(* CODESYS project para_retain.20190301.5.project

Project tree, tasks and I/O mapping:
  MIC7001 : Changsha Xiangji-ARM Cortex A9(xilinx zynq7000)-linux, Changsha Xiangji Hiden Technology Co.Ltd, version 3.5.10.40
    application Application
      libraries: CAA Types Extern, 3.5.10.0 (CAA Technical Workgroup); VisuDialogs, * (System); CAA Real Time Clock Extern, 3.5.10.0 (CAA Technical Workgroup); CAA Callback Extern, 3.5.11.0 (CAA Technical Workgroup); CAA Can Low Level Extern, 3.5.11.0 (CAA Technical Workgroup); CAA Can Low Level Imp Extern, 3.5.11.0 (CAA Technical Workgroup); SysMem, 3.5.12.0 (System); CAA Net Base Services, 3.5.12.0 (CAA Technical Workgroup); Standard, 3.5.12.0 (System); CAA SerialCom, 3.5.12.0 (CAA Technical Workgroup); CAA File, 3.5.12.0 (CAA Technical Workgroup); CAA DTUtil Extern, 3.5.12.0 (CAA Technical Workgroup); SysFile, 3.5.9.0 (System); SysTypes2 Interfaces, * (System)
      task Task (cyclic, interval 50 ms, priority 10) calls prg_main
      task VISU_TASK (cyclic, interval 100 ms, priority 31) calls VisuElems.Visu_Prg
      parameters/
        function block FB_PARA_REAL [ST]: clear_all, rd_all, wr_all, chk_chg
        data type DUT_PARA_REAL
        data type DUT_PARA_DINT
        function block FB_PARA_DINT [ST]: clear_all, rd_all, wr_all, chk_chg
      visualisation main
      program prg_main [ST]
      global variables GVL
    SoftMotion General Axis Pool
    IoDrvMIC7001 : IoDrvMIC7001, Cyber-MI, version 19.1.1
        unmapped channels: Ai00@C16, Ai01@C28, Ai02@C17, Ai03@C29, Ai04@C30, Ai05@C19, Ai06@C31, Ai07@C20, Ai08@C18, Ai09@D18, Ai10@D20, Ai11@D31, Ai12@D19, Ai13@D30, Ai14@D29, Ai15@D17, Ai16@D28, Ai17@D16, Ai18-Do00@C25, Ai19-Do01@C24, Ai20-Do02@C13, Ai21-Do03@C01, Ai22-Do04@C03, Ai23-Do05@C04, Ai24-Do06@C05, Ai25-Do07@C06, Ai26-Do08@C08, Ai27-Do09@C09, Ai28-Do10@C10, Ai29-Do11@C11, Ai30-Do12@D34, Ai31-Do13@D35, Ai32-Do14@D23, Ai33-Do15@D12, Ai34-Do16@D10, Ai35-Do17@D09, Ai36-Do18@D08, Ai37-Do19@D07, Ai38-Do20@D05, Ai39-Do21@D04,
          Ai40-Do22@D03, Ai41-Do23@D02, Ai42-Do24@C23, Ai43-Do25@C35, Ai44-Do26@D24, Ai45-Do27@D13, Ai46-Ao00@C22, Ai47-Ao01@D14, Ai48_Pi02, Ai49_Out5V, Ai50_VCC, Ai51_VCC_L, Ai52_VCC_R, Ai53_Pwm-i0, Ai54_Pwm-i1, Ai55_Pwm-i2, Ai56_Pwm-i3, Ai57_CPU-T, Ai58_G-x, Ai59_G-y, Ai60_G-z, Ai61-reserved, Ai62-IO-cntr, Ai63-CDS-cntr, Di00-Ai00@C16, Di01-Ai01@C28, Di02-Ai02@C17, Di03-Ai03@C29, Di04-Ai04@C30, Di05-Ai05@C19, Di06-Ai06@C31, Di07-Ai07@C20, Di08-Ai08@C18, Di09-Ai09@D18, Di10-Ai10@D20, Di11-Ai11@D31, Di12-Ai12@D19, Di13-Ai13@D30, Di14-Ai14@D29, Di15-Ai15@D17,
          Di16-Ai16@D28, Di17-Ai17@D16, Di18-Ai18@C25, Di19-Ai19@C24, Di20-Ai20@C13, Di21-Ai21@C01, Di22-Ai22@C03, Di23-Ai23@C04, Di24-Ai24@C05, Di25-Ai25@C06, Di26-Ai26@C08, Di27-Ai27@C09, Di28-Ai28@C10, Di29-Ai29@C11, Di30-Ai30@D34, Di31-Ai31@D35, Di32-Ai32@D23, Di33-Ai33@D12, Di34-Ai34@D10, Di35-Ai35@D09, Di36-Ai36@D08, Di37-Ai37@D07, Di38-Ai38@D05, Di39-Ai39@D04, Di40-Ai40@D03, Di41-Ai41@D02, Di42-Ai42@C23, Di43-Ai43@C35, Di44-Ai44@D24, Di45-Ai45@D13, Di46-Ai46@C22, Di47-Ai47@D14, Di48-Pi00@C15, Di49-Pi01@C14, Di50-Pi02@D22, Di51-Pi03@D21, Di52-reserved, Di53-reserved, Di54-reserved, Di55-reserved,
          Di56-reserved, Di57-reserved, Di58-reserved, Di59-reserved, Di60-reserved, Di61-reserved, Di62-reserved, Di63-reserved, Pi00-Di48@C15, Pi01-Di49@C14, Pi02-Di50@D22, Pi03-Di51@D21, Do00-Ai18@C25, Do01-Ai19@C24, Do02-Ai20@C13, Do03-Ai21@C01, Do04-Ai22@C03, Do05-Ai23@C04, Do06-Ai24@C05, Do07-Ai25@C06, Do08-Ai26@C08, Do09-Ai27@C09, Do10-Ai28@C10, Do11-Ai29@C11, Do12-Ai30@D34, Do13-Ai31@D35, Do14-Ai32@D23, Do15-Ai33@D12, Do16-Ai34@D10, Do17-Ai35@D09, Do18-Ai36@D08, Do19-Ai37@D07, Do20-Ai38@D05, Do21-Ai39@D04, Do22-Ai40@D03, Do23-Ai41@D02, Do24-Ai42@C23, Do25-Ai43@C35, Do26-Ai44@D24, Do27-Ai45@D13,
          Do28-Pwmi00@C33, Do29-Pwmi01@C34, Do30-Pwmi02@D25, Do31-Pwmi03@D26, PWM00@C25, PWM01@C24, PWM02@C13, PWM03@C01, PWM04@C03, PWM05@C04, PWM06@C05, PWM07@C06, PWM08@C08, PWM09@C09, PWM10@C10, PWM11@C11, PWM12@D34, PWM13@D35, PWM14@D23, PWM15@D12, PWM16@D10, PWM17@D09, PWM18@D08, PWM19@D07, PWM20@D05, PWM21@D04, PWM22@D03, PWM23@D02, PWM24@C23, PWM25@C35, PWM26@D24, PWM27@D13, PWM28-Pwmi00@C33, PWM29-Pwmi01@C34, PWM30-Pwmi02@D25, PWM31-Pwmi03@D26, PWM_I_0@C33, PWM_I_1@C34, PWM_I_2@D25, PWM_I_3@D26,
          Ao00-Ai46@C22, Ao01-Ai47@D14, LED_run, LED_err, LED_usr, ctrl_ai_raw, ctrl_adjust, ctrl_adj0, ctrl_adj1, ctrl_adj2, ctrl_adj3, ctrl_adj4
  5ce3da45-db07-42e7-a21c-a00fff4ed8f6|C:\Users\Administrator\Desktop\robotview1.bmp
  5ce3da45-db07-42e7-a21c-a00fff4ed8f6|C:\Users\Administrator\Desktop\robotview2.bmp
  text list GlobalTextList
  5ce3da45-db07-42e7-a21c-a00fff4ed8f6|C:\Users\Administrator\Desktop\1129.bmp
  5ce3da45-db07-42e7-a21c-a00fff4ed8f6|C:\Users\Administrator\Desktop\robotview0.bmp
*)

// MIC7001/Application/parameters/DUT_PARA_REAL
TYPE DUT_PARA_REAL :
STRUCT
	num:UINT := 256; //可根据需要设置总数量，最后一个为校验和，不可用
	para:ARRAY[1..256] OF REAL;  //三行中的总数量需要严格一致
	old_val:ARRAY[1..256] OF REAL; //三行中的总数量需要严格一致
	filename :STRING := 'mic_real.txt';  
END_STRUCT
END_TYPE

// MIC7001/Application/parameters/DUT_PARA_DINT
TYPE DUT_PARA_DINT :
STRUCT
	num:UINT := 256;  //可根据需要设置总数量，最后一个为校验和，不可用
	para:ARRAY[1..256] OF DINT;  //三行中的总数量需要严格一致
	old_val:ARRAY[1..256] OF DINT; //三行中的总数量需要严格一致
	filename :STRING := 'mic_dint.txt';  
END_STRUCT
END_TYPE

// MIC7001/Application/GVL
VAR_GLOBAL
	
END_VAR

// MIC7001/Application/prg_main
PROGRAM prg_main  //主控制程序
VAR

	para_real:DUT_PARA_REAL;
	myReal:FB_PARA_REAL := (enable := TRUE, pPara := ADR(para_real));
	
	para_dint:DUT_PARA_DINT;
	myDint:FB_PARA_DINT := (enable := TRUE, pPara := ADR(para_dint));

	rPara :REAL;
	rPara2 :REAL;
	
	rDint:DINT;
	rDint2:DINT;
END_VAR

//浮点数 参数
myReal(enable := TRUE, pPara := ADR(para_real));
//设置参数
myReal.pPara^.para[3] := 1234.56;
//读取参数
rPara := myReal.pPara^.para[3];
rPara2 := myReal.pPara^.para[4];

(*******************************************)
//整数参数
myDint(enable := TRUE, pPara := ADR(para_dint));
//设置参数
myDint.pPara^.para[3] := 1234;
//读取参数
rDint := myDint.pPara^.para[3];
rDint2 := myDint.pPara^.para[4];

END_PROGRAM

// MIC7001/Application/parameters/FB_PARA_REAL
FUNCTION_BLOCK FB_PARA_REAL
VAR_INPUT
	enable:BOOL := FALSE;
	clear:BOOL := FALSE;
	pPara:POINTER TO DUT_PARA_REAL;
END_VAR

VAR_OUTPUT
	ok:BOOL := FALSE;
	zero:BOOL := FALSE;
END_VAR

VAR
	hFile: RTS_IEC_HANDLE := 0;
	sync:BOOL := FALSE;  
	stat:UINT:= 0;
	
	i :UINT;
	str:STRING(1024);
END_VAR


IF NOT enable OR pPara^.num < 1 THEN
	stat := 0;
	RETURN;
END_IF

CASE stat OF
	0:  //init
		IF rd_all(pPara^.filename)	THEN 
			zero := FALSE;
			stat := 10;
		ELSE
			clear_all();
			IF wr_all(pPara^.filename) THEN
				zero := TRUE;
				stat := 10;
			END_IF
		END_IF
	
	10: // normal
		IF chk_chg() THEN
			ok := FALSE;
			IF wr_all(pPara^.filename) THEN
				ok := TRUE;
				zero := FALSE;
			END_IF
		END_IF	
		
		IF clear THEN
			clear_all();
			IF wr_all(pPara^.filename) THEN
				zero := TRUE;
			END_IF
		END_IF
END_CASE

METHOD clear_all : bool
VAR_INPUT
	
END_VAR
FOR i := 1 TO pPara^.num DO
	pPara^.para[i] := 0.0;
	pPara^.old_val[i] := 0.0;
END_FOR

clear_all := TRUE;
END_METHOD

METHOD rd_all : bool
VAR_INPUT
	filename:STRING(256);
END_VAR

VAR
	iNumber:INT;
	udiByteRead:LWORD;
	udiPos:UDINT;
	udiOpenError: RTS_IEC_RESULT;
	udiReadError: RTS_IEC_RESULT;
	str: STRING(255);
	ulOffset:DWORD;
	batch: BOOL;
	check_sum :REAL;
END_VAR
rd_all := FALSE;

hFile := sysfileopen(szFile := filename, am := sysfile.AM_READ, pResult:= ADR(udiOpenError));
IF hFile = RTS_INVALID_HANDLE THEN
	RETURN;
END_IF

ulOffset := 0;
batch := TRUE;

check_sum := 0.0;
FOR i := 1 TO pPara^.num DO
	IF udiByteRead < 50 AND batch THEN
		udiPos := SysFileSetPos(hFile:=hFile, ulOffset := ulOffset);
		udiByteRead := sysfile.SysFileRead(hfile := hFile,pbyBuffer := ADR(str), ulSize := 255 , pResult := ADR(udiReadError));
		IF udiByteRead < 255 THEN
			batch := FALSE;
		END_IF
	END_IF
	IF udiByteRead < 1 THEN  //读取失败
		sysfile.SysFileClose(hFile := hFile);
		RETURN;
	END_IF

	iNumber := find(str, '$N');
	IF iNumber < 2 THEN
		sysfile.SysFileClose(hFile := hFile);
		RETURN;
	END_IF
	
	pPara^.para[i] := STRING_TO_REAL(left(str,iNumber-1));
	str := delete(str, iNumber,1);
	pPara^.old_val[i] := pPara^.para[i];
	
	udiByteRead := udiByteRead - ANY_TO_LWORD(iNumber);
	ulOffset := ulOffset + ANY_TO_DWORD(iNumber);

	IF i = pPara^.num THEN
		IF ABS(check_sum-pPara^.para[i]) > 0.01 THEN
			RETURN;  //error
		END_IF
	ELSE
		check_sum := check_sum + pPara^.para[i];
	END_IF
END_FOR

sysfile.SysFileClose(hFile := hFile);
rd_all := TRUE;
END_METHOD

METHOD wr_all : bool
VAR_INPUT
	filename:STRING(256);
END_VAR

VAR
	iNumber:INT;
	udiByteWrite:LWORD;
	udiPos:UDINT;
	udiOpenError: RTS_IEC_RESULT;
	udiWriteError: RTS_IEC_RESULT;
	str_size:DWORD;
	check_sum: REAL;
END_VAR
wr_all := FALSE;
hFile := sysfileopen(szFile := filename, am := sysfile.AM_WRITE, pResult := ADR(udiOpenError));
IF hFile = RTS_INVALID_HANDLE THEN
	RETURN;
END_IF

udiPos := SysFileSetPos(hFile:=hFile, ulOffset := 0);

check_sum := 0.0;
str:= ANY_TO_STRING('');
FOR i := 1 TO pPara^.num DO
	IF i = pPara^.num THEN  //the last val, check_sum
		pPara^.para[i] := check_sum;
	ELSE
		check_sum := check_sum + pPara^.para[i];
	END_IF	
	str := concat(str, ANY_TO_STRING(pPara^.para[i]));
	str := concat(str, ANY_TO_STRING('$N'));
	str_size := ANY_TO_DWORD(len(str));
	IF str_size > 200 THEN
		udiByteWrite := sysfile.SysFileWrite(hFile := hFile,pbyBuffer := ADR(str),ulSize := str_size, pResult := ADR(udiWriteError));
		IF udiByteWrite = str_size THEN
			str := '';
		END_IF
	END_IF	
END_FOR
udiByteWrite := sysfile.SysFileWrite(hFile := hFile,pbyBuffer := ADR(str),ulSize := str_size, pResult := ADR(udiWriteError));
	
IF udiByteWrite <> str_size THEN
	sysfile.SysFileClose(hFile);
	RETURN;
END_IF
sysfile.SysFileClose(hFile);
	
FOR i := 1 TO pPara^.num DO
	pPara^.old_val[i] := pPara^.para[i];
END_FOR

hFile := 0;

wr_all := TRUE;
END_METHOD

METHOD chk_chg : bool
VAR_INPUT
END_VAR

VAR
	i :UINT;
END_VAR
chk_chg := TRUE;

FOR i := 1 TO pPara^.num  DO
	IF pPara^.para[i] <> pPara^.old_val[i] THEN
		RETURN;
	END_IF
END_FOR

chk_chg := FALSE;
END_METHOD

END_FUNCTION_BLOCK

// MIC7001/Application/parameters/FB_PARA_DINT
FUNCTION_BLOCK FB_PARA_DINT
VAR_INPUT
	enable:BOOL := FALSE;
	clear:BOOL := FALSE;
	pPara:POINTER TO DUT_PARA_DINT;
END_VAR

VAR_OUTPUT
	ok:BOOL := FALSE;
	zero:BOOL := FALSE;
END_VAR

VAR
	hFile: RTS_IEC_HANDLE := 0;
	sync:BOOL := FALSE;  
	stat:UINT:= 0;
	
	i :UINT;
END_VAR


IF NOT enable OR pPara^.num < 1 THEN
	stat := 0;
	RETURN;
END_IF

CASE stat OF
	0:  //init
		IF rd_all(pPara^.filename)	THEN 
			zero := FALSE;
			ok := TRUE;
			stat := 10;
		ELSE
			clear_all();
			IF wr_all(pPara^.filename) THEN
				zero := TRUE;
				ok := FALSE;
				stat := 10;
			END_IF
		END_IF
	
	10: // normal
		IF chk_chg() THEN
			ok := FALSE;
			IF wr_all(pPara^.filename) THEN
				ok := TRUE;
				zero := FALSE;
			END_IF
		END_IF	
		
		IF clear THEN
			clear_all();
			IF wr_all(pPara^.filename) THEN
				zero := TRUE;
				ok := FALSE;
			END_IF
		END_IF
END_CASE

METHOD clear_all : bool
VAR_INPUT
	
END_VAR
FOR i := 1 TO pPara^.num DO
	pPara^.para[i] := 0;
	pPara^.old_val[i] := 0;
END_FOR

clear_all := TRUE;
END_METHOD

METHOD rd_all : bool
VAR_INPUT
	filename:STRING(256);
END_VAR

VAR
	iNumber:INT;
	udiByteRead:LWORD;
	udiPos:UDINT;
	udiOpenError: RTS_IEC_RESULT;
	udiReadError: RTS_IEC_RESULT;
	str: STRING(255);
	ulOffset:DWORD;
	batch: BOOL;
	check_sum: DINT;
END_VAR
rd_all := FALSE;

hFile := sysfileopen(szFile := filename, am := sysfile.AM_READ, pResult:= ADR(udiOpenError));
IF hFile = RTS_INVALID_HANDLE THEN
	RETURN;
END_IF

ulOffset := 0;
batch := TRUE;

check_sum := 0;
FOR i := 1 TO pPara^.num DO
	IF udiByteRead < 50 AND batch THEN
		udiPos := SysFileSetPos(hFile:=hFile, ulOffset := ulOffset);
		udiByteRead := sysfile.SysFileRead(hfile := hFile,pbyBuffer := ADR(str), ulSize := 255 , pResult := ADR(udiReadError));
		IF udiByteRead < 255 THEN
			batch := FALSE;
		END_IF
	END_IF
	IF udiByteRead < 1 THEN  //读取失败
		sysfile.SysFileClose(hFile := hFile);
		RETURN;
	END_IF

	iNumber := find(str, '$N');
	IF iNumber < 2 THEN
		sysfile.SysFileClose(hFile := hFile);
		RETURN;
	END_IF
	
	pPara^.para[i] := STRING_TO_DINT(left(str,iNumber-1));
	str := delete(str, iNumber,1);
	pPara^.old_val[i] := pPara^.para[i];
	
	udiByteRead := udiByteRead - ANY_TO_LWORD(iNumber);
	ulOffset := ulOffset + ANY_TO_DWORD(iNumber);

	IF i = pPara^.num THEN
		IF check_sum <> pPara^.para[i] THEN
			RETURN;  //error
		END_IF
	ELSE
		check_sum := check_sum + pPara^.para[i];
	END_IF
END_FOR

sysfile.SysFileClose(hFile := hFile);
rd_all := TRUE;
END_METHOD

METHOD wr_all : bool
VAR_INPUT
	filename:STRING(256);
END_VAR

VAR
	iNumber:INT;
	udiByteWrite:LWORD;
	udiPos:UDINT;
	udiOpenError: RTS_IEC_RESULT;
	udiWriteError: RTS_IEC_RESULT;
	str_size:DWORD;
	str: STRING(255);
	check_sum: DINT;
END_VAR
wr_all := FALSE;
hFile := sysfileopen(szFile := filename, am := sysfile.AM_WRITE, pResult := ADR(udiOpenError));
IF hFile = RTS_INVALID_HANDLE THEN
	RETURN;
END_IF

udiPos := SysFileSetPos(hFile:=hFile, ulOffset := 0);

check_sum := 0;
str:= ANY_TO_STRING('');
FOR i := 1 TO pPara^.num DO
	IF i = pPara^.num THEN  //the last val, check_sum
		pPara^.para[i] := check_sum;
	ELSE
		check_sum := check_sum + pPara^.para[i];
	END_IF
	str := concat(str, ANY_TO_STRING(pPara^.para[i]));
	str := concat(str, ANY_TO_STRING('$N'));
	str_size := ANY_TO_DWORD(len(str));
	IF str_size > 200 THEN
		udiByteWrite := sysfile.SysFileWrite(hFile := hFile,pbyBuffer := ADR(str),ulSize := str_size, pResult := ADR(udiWriteError));
		IF udiByteWrite = str_size THEN
			str := '';
		END_IF
	END_IF	
END_FOR
udiByteWrite := sysfile.SysFileWrite(hFile := hFile,pbyBuffer := ADR(str),ulSize := str_size, pResult := ADR(udiWriteError));
	
IF udiByteWrite <> str_size THEN
	sysfile.SysFileClose(hFile);
	RETURN;
END_IF
sysfile.SysFileClose(hFile);

	
FOR i := 1 TO pPara^.num DO
	pPara^.old_val[i] := pPara^.para[i];
END_FOR

hFile := 0;

wr_all := TRUE;
END_METHOD

METHOD chk_chg : bool
VAR_INPUT
END_VAR

VAR
	i :UINT;
END_VAR
chk_chg := TRUE;

FOR i := 1 TO pPara^.num  DO
	IF pPara^.para[i] <> pPara^.old_val[i] THEN
		RETURN;
	END_IF
END_FOR

chk_chg := FALSE;
END_METHOD

END_FUNCTION_BLOCK

// MIC7001/Application/main
VISUALIZATION main  // 2x2
END_VISUALIZATION
